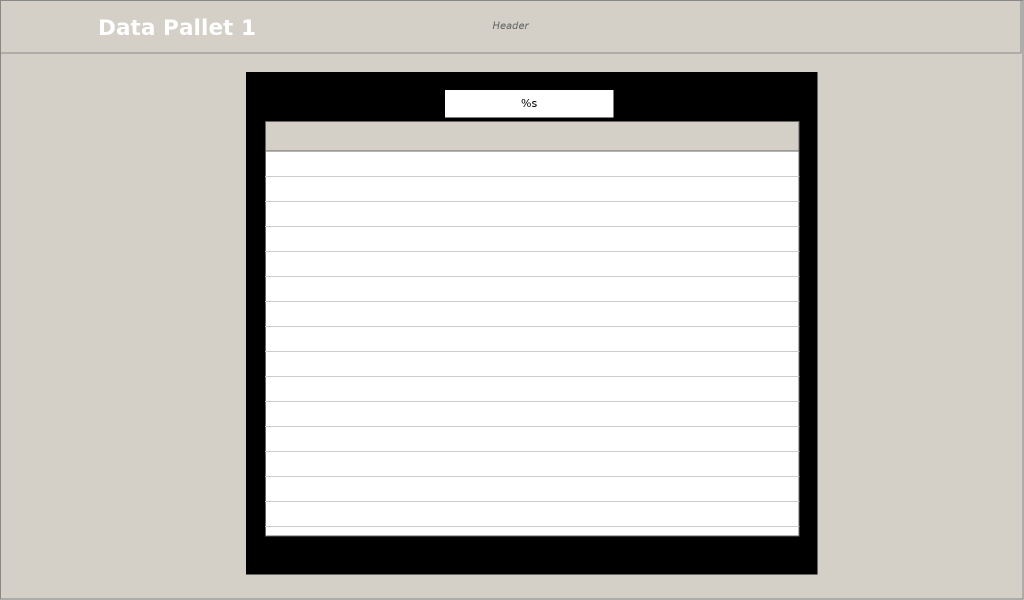
VISUALIZATION DataPallet1  // 1024x600
    Frame (0,-2 1021x55)
        shows Header()
    RoundedRectangle (246,72 571x502)
    Label (95,15 250x25), "Data Pallet 1"
    Table (265,121 534x415), data array: Status_GVL.arDataPallet1
        p3854506369: Status_GVL.arDataPallet1[INDEX].BarcodePallet
        p1892666644: Status_GVL.arDataPallet1[INDEX].BarcodePalletTime
        p338671338: Status_GVL.arPalletizingBuffer[1].EANVariant
        p2170511999: Status_GVL.arPalletizingBuffer[1].CodeVariant
        p3723444502: Status_GVL.arPalletizingBuffer[1].ProductDescription
        p1218418051: Status_GVL.arPalletizingBuffer[1].PalletCreationDate
        p746581629: Status_GVL.arPalletizingBuffer[1].BarcodeProduct
        p3104783080: Status_GVL.arPalletizingBuffer[1].BarcodeProductTime
    RoundedRectangle (444,89 170x29), "%s", text variable: Status_GVL.arPalletID[1]
END_VISUALIZATION

(* stored: Version 1.1.0.1, ProductVersion 3.1.4024.12
   Visu DataPallet1: Id {b614c883-52e7-4db6-9b9d-5a7f392514ac} *)
